% RSLogix 500 project timer question 2.RSS, saved by version 8.30.00.15 %
PROJECT "UNTITLED"    % processor: MicroLogix 1000 %

PROGRAM FILES
  LAD 2 "MAIN_PROG"  11 rungs
  LAD 3 "USER_FAULT"  1 rungs
  LAD 4 "HSC_INT"  1 rungs
  LAD 5 "STI_INT"  1 rungs
  LAD 6, 7, 8, 9, 10, 11, 12, 13, 14, 15, 16: only END

DATA FILES
  O0 OUTPUT  1 elements
  I1 INPUT  2 elements
  S2 STATUS  33 elements
  B3 BINARY  32 elements
  T4 TIMER  40 elements
  C5 COUNTER  32 elements
  R6 CONTROL  16 elements
  N7 INTEGER  105 elements

LADDER 2 "MAIN_PROG"
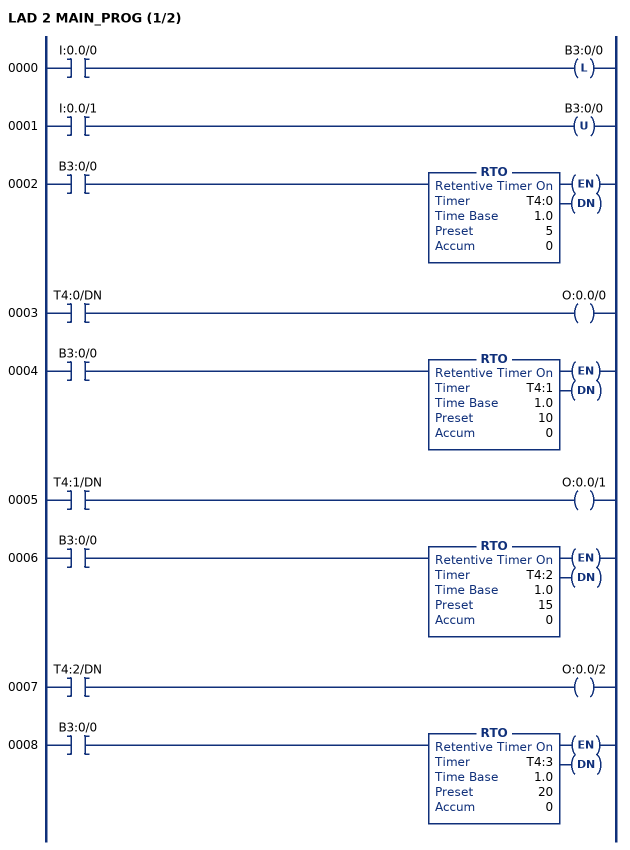
% Rung: 0 %
SOR XIC I:0.0/0 OTL B3:0/0 EOR
% Rung: 1 %
SOR XIC I:0.0/1 OTU B3:0/0 EOR
% Rung: 2 %
SOR XIC B3:0/0 RTO T4:0 1.0 5 0 EOR
% Rung: 3 %
SOR XIC T4:0/DN OTE O:0.0/0 EOR
% Rung: 4 %
SOR XIC B3:0/0 RTO T4:1 1.0 10 0 EOR
% Rung: 5 %
SOR XIC T4:1/DN OTE O:0.0/1 EOR
% Rung: 6 %
SOR XIC B3:0/0 RTO T4:2 1.0 15 0 EOR
% Rung: 7 %
SOR XIC T4:2/DN OTE O:0.0/2 EOR
% Rung: 8 %
SOR XIC B3:0/0 RTO T4:3 1.0 20 0 EOR

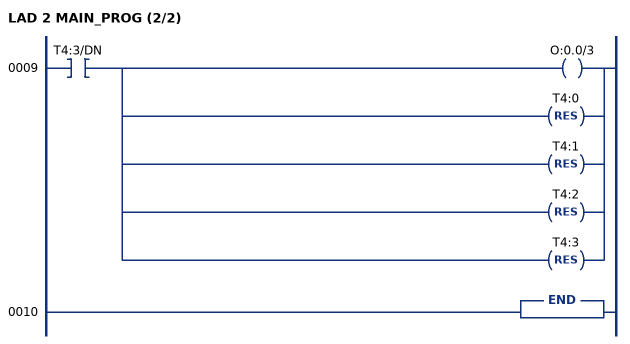
% Rung: 9 %
SOR XIC T4:3/DN BST BST BST BST OTE O:0.0/3 NXB RES T4:0 BND NXB RES T4:1 BND NXB RES T4:2 BND NXB RES T4:3 BND EOR
% Rung: 10 %
SOR END EOR

DATA TABLE (non-zero values as saved)
DATA T4
% .PRE .ACC %
% T4:0 % 5 0
% T4:1 % 10 0
% T4:2 % 15 0
% T4:3 % 20 0
